{attribute 'qualified_only'}
{attribute 'strict'}
{attribute 'to_string'}
TYPE E_APP_CHECK :
(
  NULL,

  POINTER_CTRL_INVALID                := 9000,
  POINTER_STATE_INVALID,
  REFERENCE_INSTANCE_CONTROL_INVALID,
  REFERENCE_INSTANCE_STATE_INVALID,

	POINTER_TRANSPORT_CTRL_INVALID      := 9100,
	POINTER_TRANSPORT_STATE_INVALID     := 9200,
	POINTER_COLLECTOR_ITF_INVALID       := 9300,
  REFERENCE_PROCESS_LIST_ITF_INVALID  := 9400,

  CHECK_DONE := 10000

)UINT;
END_TYPE

(* stored: Version 1.1.0.1, ProductVersion 3.1.4026.13
   DUT E_APP_CHECK: Id {def9ba09-68fc-4415-88b5-17e7f5e33a36} *)
